FUNCTION_BLOCK FB_AtomicMass_Test EXTENDS TcUnit.FB_TestSuite
VAR
    nTestID : INT;
END_VAR


nTestID := 0;

TestInvalidElementExpectNotFoundAnd0AtomicMass(
    sName := 'INVALID'
);

TestLookupInvalidElementExpectNotFoundAnd0AtomicMass(
    sName := 'INVALID'
);

TestValidElementExpectFoundAndCorrectAtomicMass(
    sName := 'Be',
    fExpectedMass := 9.012182
);

TestLookupValidElementExpectFoundAndCorrectAtomicMass(
    sName := 'Be',
    fExpectedMass := 9.012182
);

TestValidElementExpectFoundAndCorrectAtomicMass(
    sName := 'H',
    fExpectedMass := 1.00794
);

TestLookupValidElementExpectFoundAndCorrectAtomicMass(
    sName := 'H',
    fExpectedMass := 1.00794
);

TestValidElementExpectFoundAndCorrectAtomicMass(
    sName := 'Ca',
    fExpectedMass := 40.078
);

TestLookupValidElementExpectFoundAndCorrectAtomicMass(
    sName := 'Ca',
    fExpectedMass := 40.078
);

TestValidElementExpectFoundAndCorrectAtomicMass(
    sName := 'Lr',
    fExpectedMass := 262
);

TestLookupValidElementExpectFoundAndCorrectAtomicMass(
    sName := 'Lr',
    fExpectedMass := 262
);

TestValidElementExpectFoundAndCorrectAtomicMass(
    sName := 'Nb',
    fExpectedMass := 92.90638
);

TestLookupValidElementExpectFoundAndCorrectAtomicMass(
    sName := 'Nb',
    fExpectedMass := 92.90638
);


METHOD TestInvalidElementExpectNotFoundAnd0AtomicMass
VAR_INPUT
    sName : STRING;
END_VAR
VAR
    fbAtomicMass : FB_AtomicMass;
END_VAR

TEST(CONCAT('TestInvalidElementExpectNotFoundAnd0AtomicMass ID: ',
    INT_TO_STRING(nTestID))
);

fbAtomicMass(
    sName := sName,
    bFound =>,
    fValue =>,
);

AssertFalse(
    Condition := fbAtomicMass.bFound,
    Message := 'Expected bFound bit to be false but it was true.'
);

AssertTrue(
    Condition := fbAtomicMass.GetError(),
    Message := 'Expected bError bit to be true but it was false.'
);

AssertFalse(
    Condition := fbAtomicMass.GetErrorMsg() = '',
    Message := 'Expected there to be an error message but there was none.'
);

AssertTrue(
    Condition := fbAtomicMass.fValue = 0.0,
    Message := CONCAT('Expected atomic mass to be 0.0 but it was [',
        CONCAT(LREAL_TO_STRING(fbAtomicMass.fValue),
        '].'))
);

TEST_FINISHED();

nTestID := nTestID + 1;
END_METHOD


METHOD TestLookupInvalidElementExpectNotFoundAnd0AtomicMass
VAR_INPUT
    sName : STRING;
END_VAR
VAR
    fValue : LREAL;
    fbAtomicMass : FB_AtomicMass;
END_VAR

TEST(CONCAT('TestLookupInvalidElementExpectNotFoundAnd0AtomicMass ID: ',
    INT_TO_STRING(nTestID))
);

fValue := fbAtomicMass.Lookup(sLookup := sName);

AssertTrue(
    Condition := fbAtomicMass.GetError(),
    Message := 'Expected bError bit to be true but it was false.'
);

AssertFalse(
    Condition := fbAtomicMass.GetErrorMsg() = '',
    Message := 'Expected there to be an error message but there was none.'
);

AssertTrue(
    Condition := fValue = 0.0,
    Message := CONCAT('Expected atomic mass to be 0 but it was [',
        CONCAT(LREAL_TO_STRING(fValue),
        '].'))
);

TEST_FINISHED();

nTestID := nTestID + 1;
END_METHOD


METHOD TestLookupValidElementExpectFoundAndCorrectAtomicMass
VAR_INPUT
    sName : STRING;
    fExpectedMass : LREAL;
END_VAR
VAR
    fValue : LREAL;
    fbAtomicMass : FB_AtomicMass;
END_VAR

TEST(CONCAT('TestLookupValidElementExpectFoundAndCorrectAtomicMass ID: ',
    INT_TO_STRING(nTestID))
);

fValue := fbAtomicMass.Lookup(sLookup := sName);

AssertFalse(
    Condition := fbAtomicMass.GetError(),
    Message := 'Expected bError bit to be false but it was true.'
);

AssertTrue(
    Condition := fbAtomicMass.GetErrorMsg() = '',
    Message := 'Expected there to be no error message but there was one.'
);

AssertEquals_LREAL(
    Expected := fExpectedMass,
    Actual := fValue,
    Delta := 1e-9,
    Message := CONCAT('Expected atomic mass to be [',
        CONCAT(LREAL_TO_STRING(fExpectedMass),
        CONCAT('] but it was [',
        CONCAT(LREAL_TO_STRING(fValue),
        ']'))))
);

TEST_FINISHED();

nTestID := nTestID + 1;
END_METHOD


METHOD TestValidElementExpectFoundAndCorrectAtomicMass
VAR_INPUT
    sName : STRING;
    fExpectedMass : LREAL;
END_VAR
VAR
    fbAtomicMass : FB_AtomicMass;
END_VAR

TEST(CONCAT('TestValidElementExpectFoundAndCorrectAtomicMass ID: ',
    INT_TO_STRING(nTestID))
);

fbAtomicMass(
    sName := sName,
    bFound =>,
    fValue =>,
);

AssertTrue(
    Condition := fbAtomicMass.bFound,
    Message := 'Expected bFound bit to be true but it was false.'
);

AssertFalse(
    Condition := fbAtomicMass.GetError(),
    Message := 'Expected bError bit to be false but it was true.'
);

AssertTrue(
    Condition := fbAtomicMass.GetErrorMsg() = '',
    Message := 'Expected there to be no error message but there was one.'
);

AssertEquals_LREAL(
    Expected := fExpectedMass,
    Actual := fbAtomicMass.fValue,
    Delta := 1e-9,
    Message := CONCAT('Expected atomic mass to be [',
        CONCAT(LREAL_TO_STRING(fExpectedMass),
        CONCAT('] but it was [',
        CONCAT(LREAL_TO_STRING(fbAtomicMass.fValue),
        ']'))))
);

TEST_FINISHED();

nTestID := nTestID + 1;
END_METHOD

END_FUNCTION_BLOCK

(* stored: Version 1.1.0.1
   POU FB_AtomicMass_Test: Id {941b9b80-3c86-4469-9604-bd2e5bf73994}, SpecialFunc None
   Method TestInvalidElementExpectNotFoundAnd0AtomicMass: Id {92575c6a-41a9-4729-a49c-cbfd470a3f88}
   Method TestLookupInvalidElementExpectNotFoundAnd0AtomicMass: Id {3701de71-44dc-488e-aaa0-c698ed63d352}
   Method TestLookupValidElementExpectFoundAndCorrectAtomicMass: Id {ee3c50ae-73cf-40f1-ba8e-33b5b358ad7c}
   Method TestValidElementExpectFoundAndCorrectAtomicMass: Id {94d4bf94-5ef3-417d-8329-33c523502fd4} *)
